// TIA Portal V18 export
DATA_BLOCK "DataLogWrite_DB"   // DB65
// stored: AutoNumber true, DBAccessibleFromOPCUA true, InstanceOfName DataLogWrite_SFB, OfSystemLibElement DataLogWrite, OfSystemLibVersion 1.0
"DataLogWrite_SFB"
   // VAR_INPUT
   //    REQ : Bool;
   // END_VAR
   // VAR_OUTPUT
   //    DONE : Bool;
   //    BUSY : Bool;
   //    ERROR : Bool;
   //    STATUS : Word;
   // END_VAR
   // VAR_IN_OUT
   //    ID : DWord;
   // END_VAR
BEGIN
END_DATA_BLOCK
